// TIA Portal V17 export
// export: Created 2025-03-10T13:09:53.2847665Z, ExportSetting WithDefaults, DisplayName Totally Integrated Automation Portal, DisplayVersion V17 Update 8, DisplayName TIA Portal Openness, DisplayVersion V17 Update 8, DisplayName TIA Portal Version Control Interface, DisplayVersion V17, DisplayName SINAMICS Startdrive Advanced, DisplayVersion V17 SP2, DisplayName SINAMICS Startdrive G110M, G120, G120C, G120D, G120P, G115D, DisplayVersion V17 SP2, DisplayName SINAMICS Startdrive G130, G150, S120, S150, SINAMICS MV, S210, DisplayVersion V17 SP2, DisplayName STEP 7 Professional, DisplayVersion V17 Update 8, DisplayName SINUMERIK ONE STEP 7 Toolbox, DisplayVersion V17 Update 12, DisplayName SINUMERIK 840D sl STEP 7 Toolbox, DisplayVersion V17 Update 12, DisplayName STEP 7 Safety, DisplayVersion V17 Update 6, DisplayName WinCC Advanced, DisplayVersion V17 Update 8
FUNCTION_BLOCK "FB321_CHANNEL"   // FB321, LAD
{ S7_Optimized_Access := 'FALSE' }
AUTHOR : ETXETAR
VERSION : 1.0
// stored: AutoNumber false, IsIECCheckEnabled false, SetENOAutomatically false, UDAEnableTagReadback false
   VAR_INPUT
      CHANNEL_MODE_GROUP : Int;   // CHANNEL MODE GROUP
      JERK_PARAMETERS_ENABLE { ExternalAccessible := 'False'; ExternalVisible := 'False'; ExternalWritable := 'False'} : Bool;   // JERK PARAMETERS ENABLE
      ENABLE_M01 { ExternalAccessible := 'False'; ExternalVisible := 'False'; ExternalWritable := 'False'} : Bool;   // ENABLE M01
      ENABLE_DRY_RUN_TEST_PRGM { ExternalAccessible := 'False'; ExternalVisible := 'False'; ExternalWritable := 'False'} : Bool;   // ENABLE DRY RUN TEST PRGM
      FEED_DISABLE { ExternalAccessible := 'False'; ExternalVisible := 'False'; ExternalWritable := 'False'} : Bool;   // FEED DISABLE
      ENABLE_OVERRIDE { ExternalAccessible := 'False'; ExternalVisible := 'False'; ExternalWritable := 'False'} : Bool;   // OVERRIDE 0 OR 100 =0 // OVERRIDE ENABLED =1
      ENABLE_OVERRIDE_FROM_MP_OR_HT10 { ExternalAccessible := 'False'; ExternalVisible := 'False'; ExternalWritable := 'False'} : Bool;   // ENABLE OVERRIDE FROM MAIN PANEL OR HT10, TRUE = YES, FALSE = NO (VALUE IS OBTAINED FROM AN HMI SCREEN OR ANOTHER DEVICE)
      OVERRIDE_VALUE : Byte;   // OVERRIDE VALUE
      BA3_SOFTKEYS_STOP { ExternalAccessible := 'False'; ExternalVisible := 'False'; ExternalWritable := 'False'} : Bool;   // BA3 SOFTKEYS STOP
      PROG_SLECT_FAULT_CH { ExternalAccessible := 'False'; ExternalVisible := 'False'; ExternalWritable := 'False'} : Bool;   // N.O / PROGRAM SELECTION FAULT CH
      MACHINE_IS_ALARMS : Bool;   // MACHINE IS ALARMS
      MACHINE_IS_WARNINGS : Bool;   // MACHINE IS WARNINGS
      UNIT_IS_SEOC { ExternalAccessible := 'False'; ExternalVisible := 'False'; ExternalWritable := 'False'} : Bool;   // UNIT IS SEOC
      CHANNEL_M201 { ExternalAccessible := 'False'; ExternalVisible := 'False'; ExternalWritable := 'False'} : Bool;   // CHANNEL M201
      CHANNEL_MCH_RESET : Bool;   // CHANNEL MACHINE RESET
      NC_START_DUMMY_FOR_OPT { ExternalAccessible := 'False'; ExternalVisible := 'False'; ExternalWritable := 'False'} : Bool;   // NC START DUMMY FOR OPTIMIZATION
      MPP_PUSH_BUTTON_START { ExternalAccessible := 'False'; ExternalVisible := 'False'; ExternalWritable := 'False'} : Bool;   // MPP PUSH BUTTON START
      MPP_PUSH_BUTTON_NC_START : Bool;   // MPP PUSH BUTTON NC START
      MPP_BUTTON_HOME_POS { ExternalAccessible := 'False'; ExternalVisible := 'False'; ExternalWritable := 'False'} : Bool;   // MPP BUTTON HOME POSITION
      UNIT_HOME_STEP_3 { ExternalAccessible := 'False'; ExternalVisible := 'False'; ExternalWritable := 'False'} : Bool;   // UNIT HOME STEP 3
      UNIT_CYCLE_STEP_3 { ExternalAccessible := 'False'; ExternalVisible := 'False'; ExternalWritable := 'False'} : Bool;   // UNIT CYCLE STEP 3
   END_VAR
   VAR_OUTPUT
      "CH_NOT_IN SOFT_MODE_ALARM" { ExternalAccessible := 'False'; ExternalVisible := 'False'; ExternalWritable := 'False'} : Bool;   // CHANNEL NOT IN SOFT MODE ALARM
   END_VAR
   VAR_IN_OUT
      ChannelDB : "LBP_typeChanX";
   END_VAR
   VAR DB_SPECIFIC
      CH_NOT_IN_SOFT_MODE { ExternalAccessible := 'False'; ExternalVisible := 'False'; ExternalWritable := 'False'} : Bool;   // CHANNEL NOT IN SOFT MODE
      RESET_CH { ExternalAccessible := 'False'; ExternalVisible := 'False'; ExternalWritable := 'False'} : Bool;   // RESET CHANNEL
      START_CH { ExternalAccessible := 'False'; ExternalVisible := 'False'; ExternalWritable := 'False'} : Bool;   // START CHANNEL
      RESET_AUX { ExternalAccessible := 'False'; ExternalVisible := 'False'; ExternalWritable := 'False'} : Bool;   // RESET AUX
      RESET_1 { ExternalAccessible := 'False'; ExternalVisible := 'False'; ExternalWritable := 'False'} : Bool;   // RESET 1
      RESET_2 { ExternalAccessible := 'False'; ExternalVisible := 'False'; ExternalWritable := 'False'} : Bool;   // RESET 2
      PULSE { ExternalAccessible := 'False'; ExternalVisible := 'False'; ExternalWritable := 'False'} : Bool;   // PULSE
      TIMER_CH_NOT_IN_SOFT_MODE { ExternalAccessible := 'False'; ExternalVisible := 'False'; ExternalWritable := 'False'; S7_SetPoint := 'True'} : TON_TIME;   // CHANNEL NOT IN SOFT MODE TIMER
   END_VAR
   VAR_TEMP
      DB_NUMBER : DInt;   // DB NUMBER FOR ALARM AND HELP DECODING
      CHANNEL_NUM : Int;   // CHANNEL NUMBER
   END_VAR
   // TIMER_CH_NOT_IN_SOFT_MODE.PT := T#1s;
   VAR_TEMP   // added for the SCL form of the ladder/FBD networks
      _w1 : Bool;
      _w2 : Bool;
   END_VAR
BEGIN

NETWORK
TITLE = READ INSTANCE DB
      L     DINO;
      +     10#800000;
      T     #DB_NUMBER;
//READ CHANNEL NUMBER
      L     DINO;
      L     10#320;
      -I;
      T     #CHANNEL_NUM;


REGION Network 2: ACTIVATE SINGLE BLOCK / ENABLE SINGLE BLOCK
   // Step by Step mode
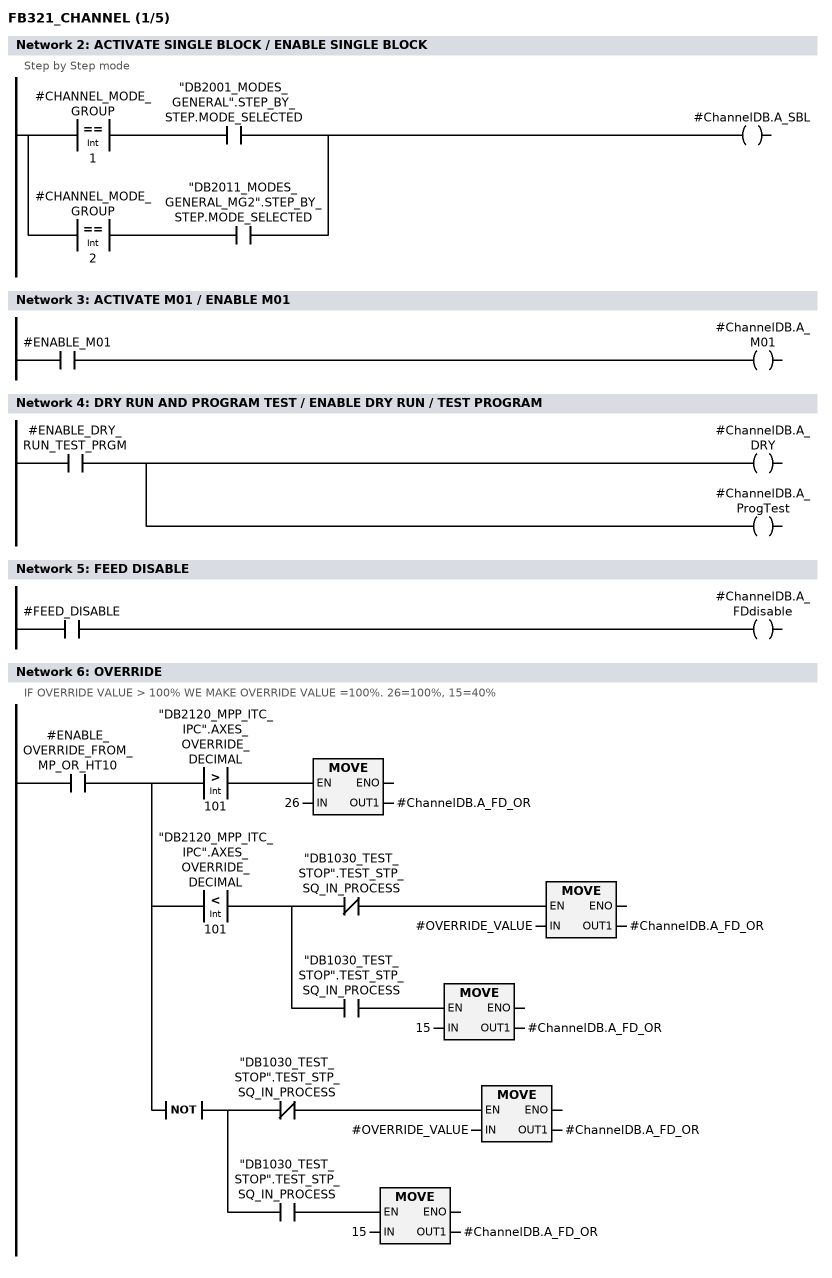
   RUNG wire#powerrail
      { S7_Templates := "SrcType := Int" } EQ_Contact(in1 := #CHANNEL_MODE_GROUP, in2 := 1)
      Contact( "DB2001_MODES_GENERAL".STEP_BY_STEP.MODE_SELECTED )
      wire#w1
      Coil( #ChannelDB.A_SBL )
   END_RUNG
   RUNG wire#powerrail
      { S7_Templates := "SrcType := Int" } EQ_Contact(in1 := #CHANNEL_MODE_GROUP, in2 := 2)
      Contact( "DB2011_MODES_GENERAL_MG2".STEP_BY_STEP.MODE_SELECTED )
   END_RUNG wire#w1
   // the same network as SCL:
   #ChannelDB.A_SBL := ((#CHANNEL_MODE_GROUP = 1) AND "DB2001_MODES_GENERAL".STEP_BY_STEP.MODE_SELECTED) OR ((#CHANNEL_MODE_GROUP = 2) AND "DB2011_MODES_GENERAL_MG2".STEP_BY_STEP.MODE_SELECTED);
END_REGION

REGION Network 3: ACTIVATE M01 / ENABLE M01
   RUNG wire#powerrail
      Contact( #ENABLE_M01 )
      Coil( #ChannelDB.A_M01 )
   END_RUNG
   // the same network as SCL:
   #ChannelDB.A_M01 := #ENABLE_M01;
END_REGION

REGION Network 4: DRY RUN AND PROGRAM TEST / ENABLE DRY RUN / TEST PROGRAM
   RUNG wire#powerrail
      Contact( #ENABLE_DRY_RUN_TEST_PRGM )
      wire#w1
      Coil( #ChannelDB.A_DRY )
   END_RUNG
   RUNG wire#w1
      Coil( #ChannelDB.A_ProgTest )
   END_RUNG
   // the same network as SCL:
   #ChannelDB.A_DRY := #ENABLE_DRY_RUN_TEST_PRGM;
   #ChannelDB.A_ProgTest := #ENABLE_DRY_RUN_TEST_PRGM;
END_REGION

REGION Network 5: FEED DISABLE
   RUNG wire#powerrail
      Contact( #FEED_DISABLE )
      Coil( #ChannelDB.A_FDdisable )
   END_RUNG
   // the same network as SCL:
   #ChannelDB.A_FDdisable := #FEED_DISABLE;
END_REGION

REGION Network 6: OVERRIDE
   // IF OVERRIDE VALUE > 100% WE MAKE OVERRIDE VALUE =100%. 26=100%, 15=40%
   RUNG wire#powerrail
      Contact( #ENABLE_OVERRIDE_FROM_MP_OR_HT10 )
      wire#w1
      { S7_Templates := "SrcType := Int" } GT_Contact(in1 := "DB2120_MPP_ITC_IPC".AXES_OVERRIDE_DECIMAL, in2 := 101)
      { S7_GenerateENO := "TRUE" } Move(in := 26, out1 => #ChannelDB.A_FD_OR)
   END_RUNG
   RUNG wire#w1
      { S7_Templates := "SrcType := Int" } LT_Contact(in1 := "DB2120_MPP_ITC_IPC".AXES_OVERRIDE_DECIMAL, in2 := 101)
      wire#w2
      I_Contact( "DB1030_TEST_STOP".TEST_STP_SQ_IN_PROCESS )
      { S7_GenerateENO := "TRUE" } Move(in := #OVERRIDE_VALUE, out1 => #ChannelDB.A_FD_OR)
   END_RUNG
   RUNG wire#w2
      Contact( "DB1030_TEST_STOP".TEST_STP_SQ_IN_PROCESS )
      { S7_GenerateENO := "TRUE" } Move(in := 15, out1 => #ChannelDB.A_FD_OR)
   END_RUNG
   RUNG wire#w1
      Not()
      wire#w3
      I_Contact( "DB1030_TEST_STOP".TEST_STP_SQ_IN_PROCESS )
      { S7_GenerateENO := "TRUE" } Move(in := #OVERRIDE_VALUE, out1 => #ChannelDB.A_FD_OR)
   END_RUNG
   RUNG wire#w3
      Contact( "DB1030_TEST_STOP".TEST_STP_SQ_IN_PROCESS )
      { S7_GenerateENO := "TRUE" } Move(in := 15, out1 => #ChannelDB.A_FD_OR)
   END_RUNG
   // the same network as SCL:
   IF #ENABLE_OVERRIDE_FROM_MP_OR_HT10 AND ("DB2120_MPP_ITC_IPC".AXES_OVERRIDE_DECIMAL > 101) THEN
       #ChannelDB.A_FD_OR := 26;
   END_IF;
   #_w1 := #ENABLE_OVERRIDE_FROM_MP_OR_HT10 AND ("DB2120_MPP_ITC_IPC".AXES_OVERRIDE_DECIMAL < 101);
   IF #_w1 AND NOT "DB1030_TEST_STOP".TEST_STP_SQ_IN_PROCESS THEN
       #ChannelDB.A_FD_OR := #OVERRIDE_VALUE;
   END_IF;
   IF #_w1 AND "DB1030_TEST_STOP".TEST_STP_SQ_IN_PROCESS THEN #ChannelDB.A_FD_OR := 15; END_IF;
   #_w2 := NOT #ENABLE_OVERRIDE_FROM_MP_OR_HT10;
   IF #_w2 AND NOT "DB1030_TEST_STOP".TEST_STP_SQ_IN_PROCESS THEN
       #ChannelDB.A_FD_OR := #OVERRIDE_VALUE;
   END_IF;
   IF #_w2 AND "DB1030_TEST_STOP".TEST_STP_SQ_IN_PROCESS THEN #ChannelDB.A_FD_OR := 15; END_IF;
END_REGION

REGION Network 7: OVERRIDE ACTIVE / FEEDRATE OVERRIDE ACTIVE
   // REMOVE DUMMY ON IF REQUIRED
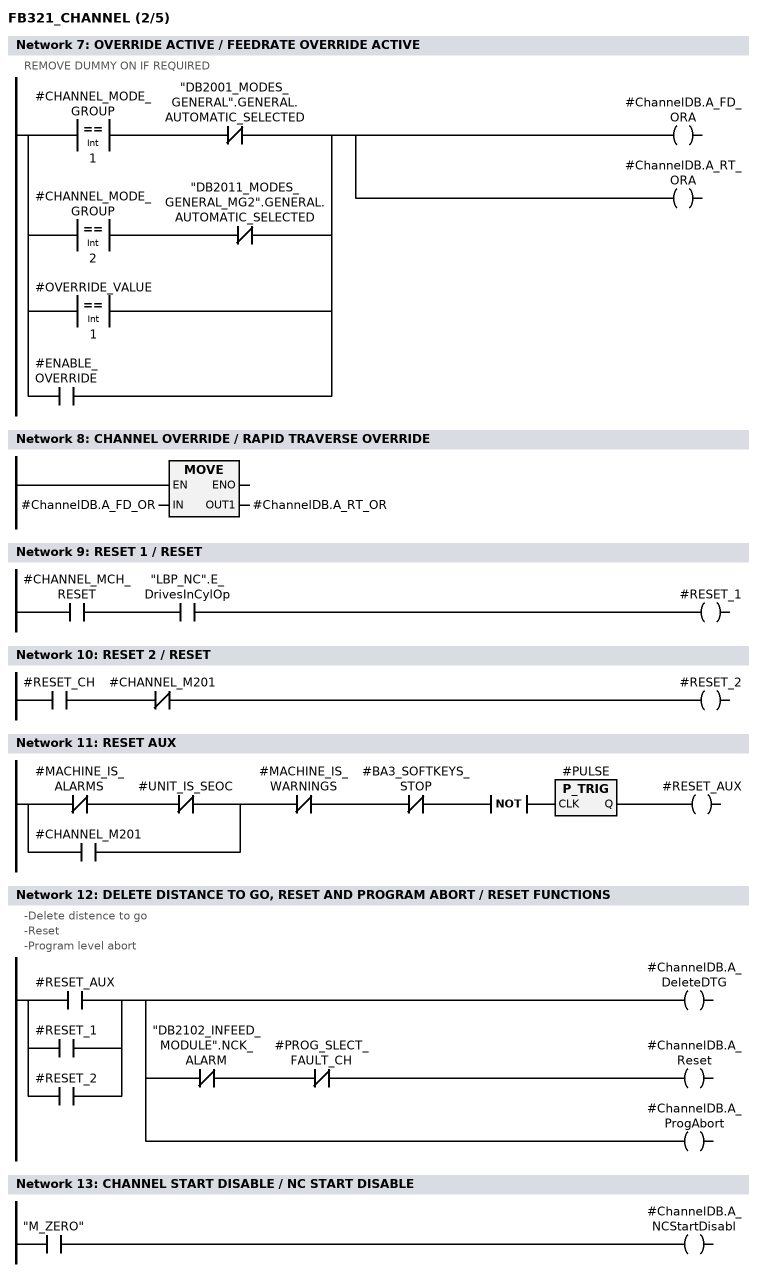
   RUNG wire#powerrail
      { S7_Templates := "SrcType := Int" } EQ_Contact(in1 := #CHANNEL_MODE_GROUP, in2 := 1)
      I_Contact( "DB2001_MODES_GENERAL".GENERAL.AUTOMATIC_SELECTED )
      wire#w1
      Coil( #ChannelDB.A_FD_ORA )
   END_RUNG
   RUNG wire#powerrail
      { S7_Templates := "SrcType := Int" } EQ_Contact(in1 := #CHANNEL_MODE_GROUP, in2 := 2)
      I_Contact( "DB2011_MODES_GENERAL_MG2".GENERAL.AUTOMATIC_SELECTED )
   END_RUNG wire#w1
   RUNG wire#powerrail
      { S7_Templates := "SrcType := Int" } EQ_Contact(in1 := #OVERRIDE_VALUE, in2 := 1)
   END_RUNG wire#w1
   RUNG wire#powerrail
      Contact( #ENABLE_OVERRIDE )
   END_RUNG wire#w1
   RUNG wire#w1
      Coil( #ChannelDB.A_RT_ORA )
   END_RUNG
   // the same network as SCL:
   #ChannelDB.A_FD_ORA := ((#CHANNEL_MODE_GROUP = 1) AND NOT "DB2001_MODES_GENERAL".GENERAL.AUTOMATIC_SELECTED) OR ((#CHANNEL_MODE_GROUP = 2) AND NOT "DB2011_MODES_GENERAL_MG2".GENERAL.AUTOMATIC_SELECTED) OR (#OVERRIDE_VALUE = 1) OR #ENABLE_OVERRIDE;
   #ChannelDB.A_RT_ORA := #ChannelDB.A_FD_ORA;
END_REGION

REGION Network 8: CHANNEL OVERRIDE / RAPID TRAVERSE OVERRIDE
   RUNG wire#powerrail
      { S7_GenerateENO := "TRUE" } Move(in := #ChannelDB.A_FD_OR, out1 => #ChannelDB.A_RT_OR)
   END_RUNG
   // the same network as SCL:
   #ChannelDB.A_RT_OR := #ChannelDB.A_FD_OR;
END_REGION

REGION Network 9: RESET 1 / RESET
   RUNG wire#powerrail
      Contact( #CHANNEL_MCH_RESET )
      Contact( "LBP_NC".E_DrivesInCylOp )
      Coil( #RESET_1 )
   END_RUNG
   // the same network as SCL:
   #RESET_1 := #CHANNEL_MCH_RESET AND "LBP_NC".E_DrivesInCylOp;
END_REGION

REGION Network 10: RESET 2 / RESET
   RUNG wire#powerrail
      Contact( #RESET_CH )
      I_Contact( #CHANNEL_M201 )
      Coil( #RESET_2 )
   END_RUNG
   // the same network as SCL:
   #RESET_2 := #RESET_CH AND NOT #CHANNEL_M201;
END_REGION

REGION Network 11: RESET AUX
   RUNG wire#powerrail
      I_Contact( #MACHINE_IS_ALARMS )
      I_Contact( #UNIT_IS_SEOC )
      wire#w1
      I_Contact( #MACHINE_IS_WARNINGS )
      I_Contact( #BA3_SOFTKEYS_STOP )
      Not()
      P_Trig( #PULSE )
      Coil( #RESET_AUX )
   END_RUNG
   RUNG wire#powerrail
      Contact( #CHANNEL_M201 )
   END_RUNG wire#w1
   // the same network as SCL:
   #_w1 := NOT (((NOT #MACHINE_IS_ALARMS AND NOT #UNIT_IS_SEOC) OR #CHANNEL_M201) AND NOT #MACHINE_IS_WARNINGS AND NOT #BA3_SOFTKEYS_STOP);
   #_w2 := #_w1 AND NOT #PULSE;   // rising edge
   #PULSE := #_w1;
   #RESET_AUX := #_w2;
END_REGION

REGION Network 12: DELETE DISTANCE TO GO, RESET AND PROGRAM ABORT / RESET FUNCTIONS
   // -Delete distence to go
   // -Reset
   // -Program level abort
   RUNG wire#powerrail
      Contact( #RESET_AUX )
      wire#w1
      Coil( #ChannelDB.A_DeleteDTG )
   END_RUNG
   RUNG wire#powerrail
      Contact( #RESET_1 )
   END_RUNG wire#w1
   RUNG wire#powerrail
      Contact( #RESET_2 )
   END_RUNG wire#w1
   RUNG wire#w1
      I_Contact( "DB2102_INFEED_MODULE".NCK_ALARM )
      I_Contact( #PROG_SLECT_FAULT_CH )
      Coil( #ChannelDB.A_Reset )
   END_RUNG
   RUNG wire#w1
      Coil( #ChannelDB.A_ProgAbort )
   END_RUNG
   // the same network as SCL:
   #ChannelDB.A_DeleteDTG := #RESET_AUX OR #RESET_1 OR #RESET_2;
   #ChannelDB.A_Reset := #ChannelDB.A_DeleteDTG AND NOT "DB2102_INFEED_MODULE".NCK_ALARM AND NOT #PROG_SLECT_FAULT_CH;
   #ChannelDB.A_ProgAbort := #ChannelDB.A_DeleteDTG;
END_REGION

REGION Network 13: CHANNEL START DISABLE / NC START DISABLE
   RUNG wire#powerrail
      Contact( "M_ZERO" )
      Coil( #ChannelDB.A_NCStartDisabl )
   END_RUNG
   // the same network as SCL:
   #ChannelDB.A_NCStartDisabl := "M_ZERO";
END_REGION

REGION Network 14: START CHANNEL / NC START
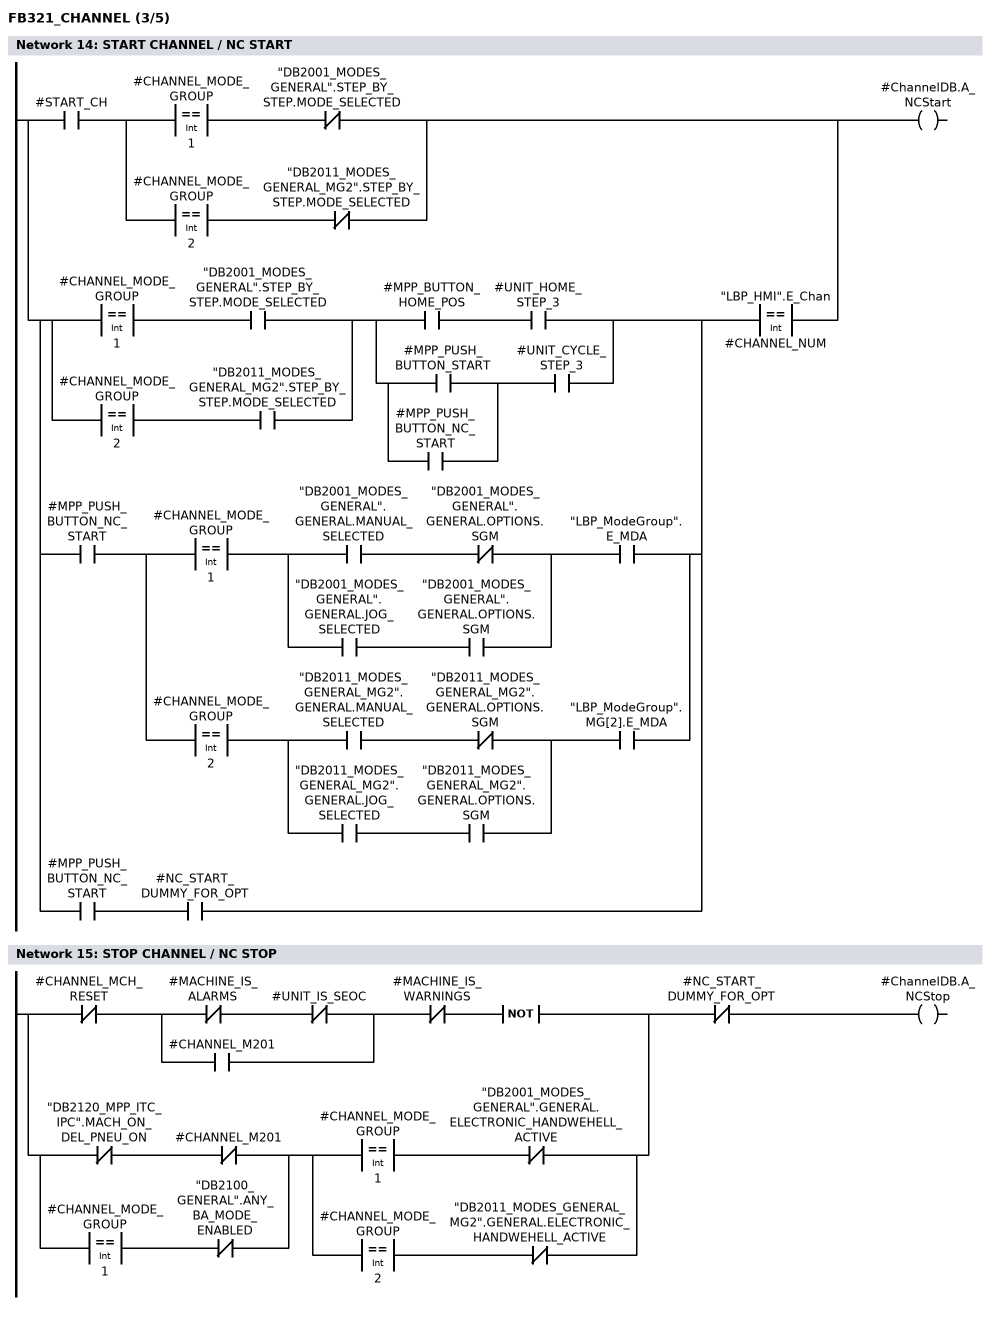
   RUNG wire#powerrail
      Contact( #START_CH )
      wire#w1
      { S7_Templates := "SrcType := Int" } EQ_Contact(in1 := #CHANNEL_MODE_GROUP, in2 := 1)
      I_Contact( "DB2001_MODES_GENERAL".STEP_BY_STEP.MODE_SELECTED )
      wire#w2
      Coil( #ChannelDB.A_NCStart )
   END_RUNG
   RUNG wire#w1
      { S7_Templates := "SrcType := Int" } EQ_Contact(in1 := #CHANNEL_MODE_GROUP, in2 := 2)
      I_Contact( "DB2011_MODES_GENERAL_MG2".STEP_BY_STEP.MODE_SELECTED )
   END_RUNG wire#w2
   RUNG wire#powerrail
      { S7_Templates := "SrcType := Int" } EQ_Contact(in1 := #CHANNEL_MODE_GROUP, in2 := 1)
      Contact( "DB2001_MODES_GENERAL".STEP_BY_STEP.MODE_SELECTED )
      wire#w3
      Contact( #MPP_BUTTON_HOME_POS )
      Contact( #UNIT_HOME_STEP_3 )
      wire#w4
      { S7_Templates := "SrcType := Int" } EQ_Contact(in1 := "LBP_HMI".E_Chan, in2 := #CHANNEL_NUM)
   END_RUNG wire#w2
   RUNG wire#powerrail
      { S7_Templates := "SrcType := Int" } EQ_Contact(in1 := #CHANNEL_MODE_GROUP, in2 := 2)
      Contact( "DB2011_MODES_GENERAL_MG2".STEP_BY_STEP.MODE_SELECTED )
   END_RUNG wire#w3
   RUNG wire#w3
      Contact( #MPP_PUSH_BUTTON_START )
      wire#w5
      Contact( #UNIT_CYCLE_STEP_3 )
   END_RUNG wire#w4
   RUNG wire#w3
      Contact( #MPP_PUSH_BUTTON_NC_START )
   END_RUNG wire#w5
   RUNG wire#powerrail
      Contact( #MPP_PUSH_BUTTON_NC_START )
      wire#w6
      { S7_Templates := "SrcType := Int" } EQ_Contact(in1 := #CHANNEL_MODE_GROUP, in2 := 1)
      wire#w7
      Contact( "DB2001_MODES_GENERAL".GENERAL.MANUAL_SELECTED )
      I_Contact( "DB2001_MODES_GENERAL".GENERAL.OPTIONS.SGM )
      wire#w8
      Contact( "LBP_ModeGroup".E_MDA )
   END_RUNG wire#w4
   RUNG wire#w7
      Contact( "DB2001_MODES_GENERAL".GENERAL.JOG_SELECTED )
      Contact( "DB2001_MODES_GENERAL".GENERAL.OPTIONS.SGM )
   END_RUNG wire#w8
   RUNG wire#w6
      { S7_Templates := "SrcType := Int" } EQ_Contact(in1 := #CHANNEL_MODE_GROUP, in2 := 2)
      wire#w9
      Contact( "DB2011_MODES_GENERAL_MG2".GENERAL.MANUAL_SELECTED )
      I_Contact( "DB2011_MODES_GENERAL_MG2".GENERAL.OPTIONS.SGM )
      wire#w10
      Contact( "LBP_ModeGroup".MG[2].E_MDA )
   END_RUNG wire#w4
   RUNG wire#w9
      Contact( "DB2011_MODES_GENERAL_MG2".GENERAL.JOG_SELECTED )
      Contact( "DB2011_MODES_GENERAL_MG2".GENERAL.OPTIONS.SGM )
   END_RUNG wire#w10
   RUNG wire#powerrail
      Contact( #MPP_PUSH_BUTTON_NC_START )
      Contact( #NC_START_DUMMY_FOR_OPT )
   END_RUNG wire#w4
   // the same network as SCL:
   #ChannelDB.A_NCStart := (#START_CH AND (((#CHANNEL_MODE_GROUP = 1) AND NOT "DB2001_MODES_GENERAL".STEP_BY_STEP.MODE_SELECTED) OR ((#CHANNEL_MODE_GROUP = 2) AND NOT "DB2011_MODES_GENERAL_MG2".STEP_BY_STEP.MODE_SELECTED))) OR ((((((#CHANNEL_MODE_GROUP = 1) AND "DB2001_MODES_GENERAL".STEP_BY_STEP.MODE_SELECTED) OR ((#CHANNEL_MODE_GROUP = 2) AND "DB2011_MODES_GENERAL_MG2".STEP_BY_STEP.MODE_SELECTED)) AND ((#MPP_BUTTON_HOME_POS AND #UNIT_HOME_STEP_3) OR ((#MPP_PUSH_BUTTON_START OR #MPP_PUSH_BUTTON_NC_START) AND #UNIT_CYCLE_STEP_3))) OR (#MPP_PUSH_BUTTON_NC_START AND (((#CHANNEL_MODE_GROUP = 1) AND (("DB2001_MODES_GENERAL".GENERAL.MANUAL_SELECTED AND NOT "DB2001_MODES_GENERAL".GENERAL.OPTIONS.SGM) OR ("DB2001_MODES_GENERAL".GENERAL.JOG_SELECTED AND "DB2001_MODES_GENERAL".GENERAL.OPTIONS.SGM)) AND "LBP_ModeGroup".E_MDA) OR ((#CHANNEL_MODE_GROUP = 2) AND (("DB2011_MODES_GENERAL_MG2".GENERAL.MANUAL_SELECTED AND NOT "DB2011_MODES_GENERAL_MG2".GENERAL.OPTIONS.SGM) OR ("DB2011_MODES_GENERAL_MG2".GENERAL.JOG_SELECTED AND "DB2011_MODES_GENERAL_MG2".GENERAL.OPTIONS.SGM)) AND "LBP_ModeGroup".MG[2].E_MDA))) OR (#MPP_PUSH_BUTTON_NC_START AND #NC_START_DUMMY_FOR_OPT)) AND ("LBP_HMI".E_Chan = #CHANNEL_NUM));
END_REGION

REGION Network 15: STOP CHANNEL / NC STOP
   RUNG wire#powerrail
      I_Contact( #CHANNEL_MCH_RESET )
      wire#w1
      I_Contact( #MACHINE_IS_ALARMS )
      I_Contact( #UNIT_IS_SEOC )
      wire#w2
      I_Contact( #MACHINE_IS_WARNINGS )
      Not()
      wire#w3
      I_Contact( #NC_START_DUMMY_FOR_OPT )
      Coil( #ChannelDB.A_NCStop )
   END_RUNG
   RUNG wire#w1
      Contact( #CHANNEL_M201 )
   END_RUNG wire#w2
   RUNG wire#powerrail
      I_Contact( "DB2120_MPP_ITC_IPC".MACH_ON_DEL_PNEU_ON )
      I_Contact( #CHANNEL_M201 )
      wire#w4
      { S7_Templates := "SrcType := Int" } EQ_Contact(in1 := #CHANNEL_MODE_GROUP, in2 := 1)
      I_Contact( "DB2001_MODES_GENERAL".GENERAL.ELECTRONIC_HANDWEHELL_ACTIVE )
   END_RUNG wire#w3
   RUNG wire#powerrail
      { S7_Templates := "SrcType := Int" } EQ_Contact(in1 := #CHANNEL_MODE_GROUP, in2 := 1)
      I_Contact( "DB2100_GENERAL".ANY_BA_MODE_ENABLED )
   END_RUNG wire#w4
   RUNG wire#w4
      { S7_Templates := "SrcType := Int" } EQ_Contact(in1 := #CHANNEL_MODE_GROUP, in2 := 2)
      I_Contact( "DB2011_MODES_GENERAL_MG2".GENERAL.ELECTRONIC_HANDWEHELL_ACTIVE )
   END_RUNG wire#w3
   // the same network as SCL:
   #ChannelDB.A_NCStop := (NOT (NOT #CHANNEL_MCH_RESET AND ((NOT #MACHINE_IS_ALARMS AND NOT #UNIT_IS_SEOC) OR #CHANNEL_M201) AND NOT #MACHINE_IS_WARNINGS) OR (((NOT "DB2120_MPP_ITC_IPC".MACH_ON_DEL_PNEU_ON AND NOT #CHANNEL_M201) OR ((#CHANNEL_MODE_GROUP = 1) AND NOT "DB2100_GENERAL".ANY_BA_MODE_ENABLED)) AND (((#CHANNEL_MODE_GROUP = 1) AND NOT "DB2001_MODES_GENERAL".GENERAL.ELECTRONIC_HANDWEHELL_ACTIVE) OR ((#CHANNEL_MODE_GROUP = 2) AND NOT "DB2011_MODES_GENERAL_MG2".GENERAL.ELECTRONIC_HANDWEHELL_ACTIVE)))) AND NOT #NC_START_DUMMY_FOR_OPT;
END_REGION

REGION Network 16: CHANNEL NOT IN SOFT MODE ALARM / SOFT MODE ACTIVE CHANNEL
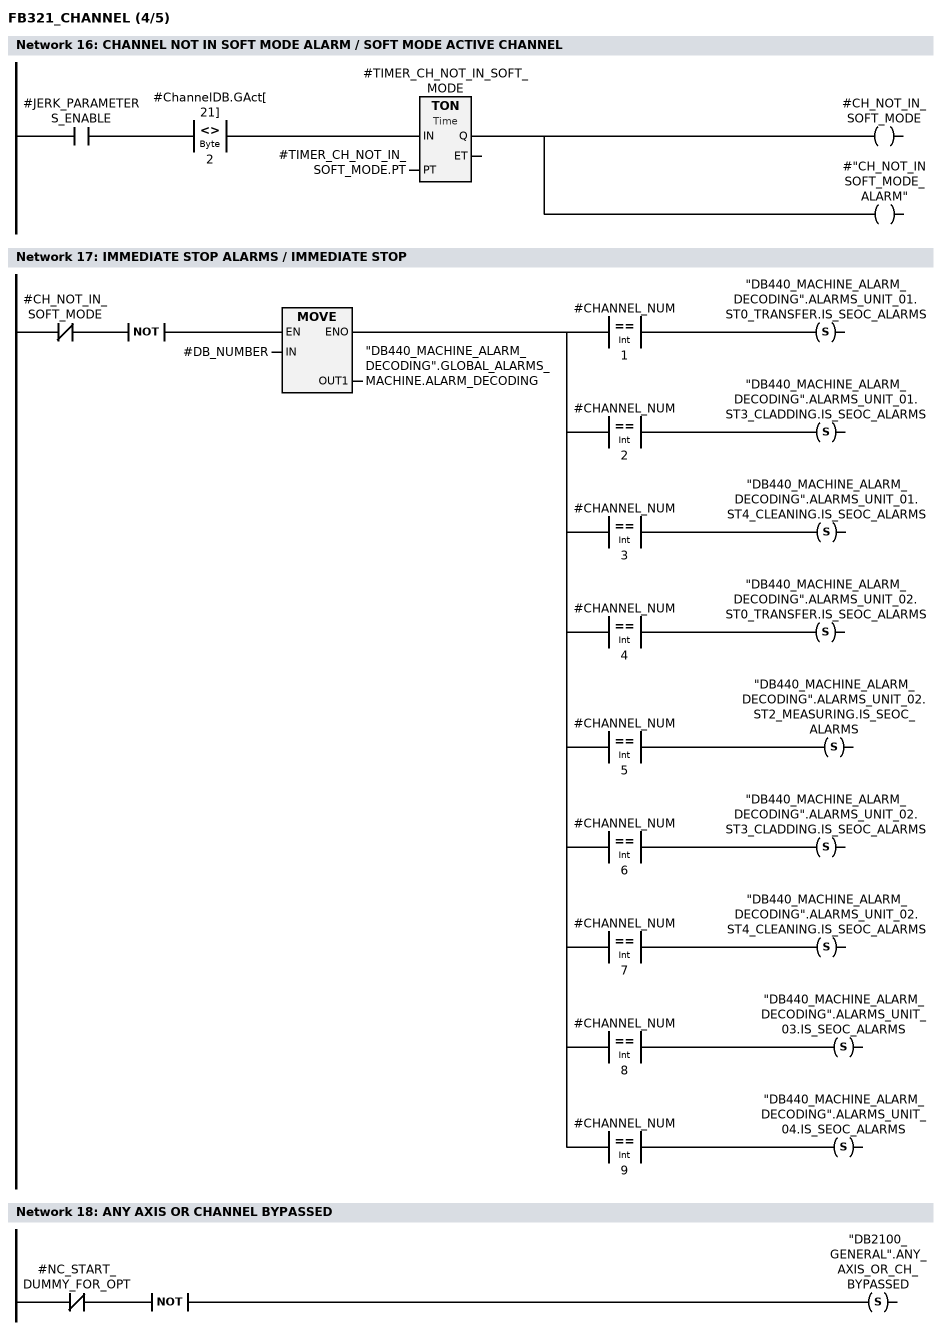
   RUNG wire#powerrail
      Contact( #JERK_PARAMETERS_ENABLE )
      { S7_Templates := "SrcType := Byte" } NE_Contact(in1 := #ChannelDB.GAct[21], in2 := 2)
      { S7_Templates := "time_type := Time" } #TIMER_CH_NOT_IN_SOFT_MODE.TON(pt := #TIMER_CH_NOT_IN_SOFT_MODE.PT, et =>)
      wire#w1
      Coil( #CH_NOT_IN_SOFT_MODE )
   END_RUNG
   RUNG wire#w1
      Coil( #"CH_NOT_IN SOFT_MODE_ALARM" )
   END_RUNG
   // the same network as SCL:
   #TIMER_CH_NOT_IN_SOFT_MODE(IN := #JERK_PARAMETERS_ENABLE AND (#ChannelDB.GAct[21] <> 2),   // TON
                           PT := #TIMER_CH_NOT_IN_SOFT_MODE.PT);
   #CH_NOT_IN_SOFT_MODE := #TIMER_CH_NOT_IN_SOFT_MODE.Q;
   #"CH_NOT_IN SOFT_MODE_ALARM" := #TIMER_CH_NOT_IN_SOFT_MODE.Q;
END_REGION

REGION Network 17: IMMEDIATE STOP ALARMS / IMMEDIATE STOP
   RUNG wire#powerrail
      I_Contact( #CH_NOT_IN_SOFT_MODE )
      Not()
      { S7_GenerateENO := "TRUE" } Move(in := #DB_NUMBER, out1 => "DB440_MACHINE_ALARM_DECODING".GLOBAL_ALARMS_MACHINE.ALARM_DECODING)
      wire#w1
      { S7_Templates := "SrcType := Int" } EQ_Contact(in1 := #CHANNEL_NUM, in2 := 1)
      S_Coil( "DB440_MACHINE_ALARM_DECODING".ALARMS_UNIT_01.ST0_TRANSFER.IS_SEOC_ALARMS )
   END_RUNG
   RUNG wire#w1
      { S7_Templates := "SrcType := Int" } EQ_Contact(in1 := #CHANNEL_NUM, in2 := 2)
      S_Coil( "DB440_MACHINE_ALARM_DECODING".ALARMS_UNIT_01.ST3_CLADDING.IS_SEOC_ALARMS )
   END_RUNG
   RUNG wire#w1
      { S7_Templates := "SrcType := Int" } EQ_Contact(in1 := #CHANNEL_NUM, in2 := 3)
      S_Coil( "DB440_MACHINE_ALARM_DECODING".ALARMS_UNIT_01.ST4_CLEANING.IS_SEOC_ALARMS )
   END_RUNG
   RUNG wire#w1
      { S7_Templates := "SrcType := Int" } EQ_Contact(in1 := #CHANNEL_NUM, in2 := 4)
      S_Coil( "DB440_MACHINE_ALARM_DECODING".ALARMS_UNIT_02.ST0_TRANSFER.IS_SEOC_ALARMS )
   END_RUNG
   RUNG wire#w1
      { S7_Templates := "SrcType := Int" } EQ_Contact(in1 := #CHANNEL_NUM, in2 := 5)
      S_Coil( "DB440_MACHINE_ALARM_DECODING".ALARMS_UNIT_02.ST2_MEASURING.IS_SEOC_ALARMS )
   END_RUNG
   RUNG wire#w1
      { S7_Templates := "SrcType := Int" } EQ_Contact(in1 := #CHANNEL_NUM, in2 := 6)
      S_Coil( "DB440_MACHINE_ALARM_DECODING".ALARMS_UNIT_02.ST3_CLADDING.IS_SEOC_ALARMS )
   END_RUNG
   RUNG wire#w1
      { S7_Templates := "SrcType := Int" } EQ_Contact(in1 := #CHANNEL_NUM, in2 := 7)
      S_Coil( "DB440_MACHINE_ALARM_DECODING".ALARMS_UNIT_02.ST4_CLEANING.IS_SEOC_ALARMS )
   END_RUNG
   RUNG wire#w1
      { S7_Templates := "SrcType := Int" } EQ_Contact(in1 := #CHANNEL_NUM, in2 := 8)
      S_Coil( "DB440_MACHINE_ALARM_DECODING".ALARMS_UNIT_03.IS_SEOC_ALARMS )
   END_RUNG
   RUNG wire#w1
      { S7_Templates := "SrcType := Int" } EQ_Contact(in1 := #CHANNEL_NUM, in2 := 9)
      S_Coil( "DB440_MACHINE_ALARM_DECODING".ALARMS_UNIT_04.IS_SEOC_ALARMS )
   END_RUNG
   // the same network as SCL:
   // ENO of a box is taken as its EN; it also drops when the box reports an error
   #_w1 := NOT (NOT #CH_NOT_IN_SOFT_MODE);
   IF #_w1 THEN "DB440_MACHINE_ALARM_DECODING".GLOBAL_ALARMS_MACHINE.ALARM_DECODING := #DB_NUMBER; END_IF;
   IF #_w1 AND (#CHANNEL_NUM = 1) THEN
       "DB440_MACHINE_ALARM_DECODING".ALARMS_UNIT_01.ST0_TRANSFER.IS_SEOC_ALARMS := TRUE;
   END_IF;
   IF #_w1 AND (#CHANNEL_NUM = 2) THEN
       "DB440_MACHINE_ALARM_DECODING".ALARMS_UNIT_01.ST3_CLADDING.IS_SEOC_ALARMS := TRUE;
   END_IF;
   IF #_w1 AND (#CHANNEL_NUM = 3) THEN
       "DB440_MACHINE_ALARM_DECODING".ALARMS_UNIT_01.ST4_CLEANING.IS_SEOC_ALARMS := TRUE;
   END_IF;
   IF #_w1 AND (#CHANNEL_NUM = 4) THEN
       "DB440_MACHINE_ALARM_DECODING".ALARMS_UNIT_02.ST0_TRANSFER.IS_SEOC_ALARMS := TRUE;
   END_IF;
   IF #_w1 AND (#CHANNEL_NUM = 5) THEN
       "DB440_MACHINE_ALARM_DECODING".ALARMS_UNIT_02.ST2_MEASURING.IS_SEOC_ALARMS := TRUE;
   END_IF;
   IF #_w1 AND (#CHANNEL_NUM = 6) THEN
       "DB440_MACHINE_ALARM_DECODING".ALARMS_UNIT_02.ST3_CLADDING.IS_SEOC_ALARMS := TRUE;
   END_IF;
   IF #_w1 AND (#CHANNEL_NUM = 7) THEN
       "DB440_MACHINE_ALARM_DECODING".ALARMS_UNIT_02.ST4_CLEANING.IS_SEOC_ALARMS := TRUE;
   END_IF;
   IF #_w1 AND (#CHANNEL_NUM = 8) THEN
       "DB440_MACHINE_ALARM_DECODING".ALARMS_UNIT_03.IS_SEOC_ALARMS := TRUE;
   END_IF;
   IF #_w1 AND (#CHANNEL_NUM = 9) THEN
       "DB440_MACHINE_ALARM_DECODING".ALARMS_UNIT_04.IS_SEOC_ALARMS := TRUE;
   END_IF;
END_REGION

REGION Network 18: ANY AXIS OR CHANNEL BYPASSED
   RUNG wire#powerrail
      I_Contact( #NC_START_DUMMY_FOR_OPT )
      Not()
      S_Coil( "DB2100_GENERAL".ANY_AXIS_OR_CH_BYPASSED )
   END_RUNG
   // the same network as SCL:
   IF NOT (NOT #NC_START_DUMMY_FOR_OPT) THEN "DB2100_GENERAL".ANY_AXIS_OR_CH_BYPASSED := TRUE; END_IF;
END_REGION

REGION Network 19: PROGRAMMING ALARM
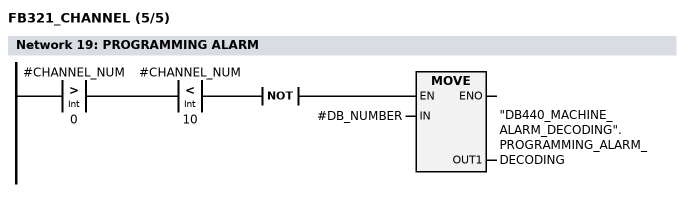
   RUNG wire#powerrail
      { S7_Templates := "SrcType := Int" } GT_Contact(in1 := #CHANNEL_NUM, in2 := 0)
      { S7_Templates := "SrcType := Int" } LT_Contact(in1 := #CHANNEL_NUM, in2 := 10)
      Not()
      Move(in := #DB_NUMBER, out1 => "DB440_MACHINE_ALARM_DECODING".PROGRAMMING_ALARM_DECODING)
   END_RUNG
   // the same network as SCL:
   IF NOT ((#CHANNEL_NUM > 0) AND (#CHANNEL_NUM < 10)) THEN
       "DB440_MACHINE_ALARM_DECODING".PROGRAMMING_ALARM_DECODING := #DB_NUMBER;
   END_IF;
END_REGION
END_FUNCTION_BLOCK
